// TwinCAT 3 PLC project PLC1
// ProgramVersion: 3.1.4024.0
// libraries:
//   Tc2_Standard, * (Beckhoff Automation GmbH)
//   Tc2_System, * (Beckhoff Automation GmbH)
//   Tc3_Module, * (Beckhoff Automation GmbH)
// project tree:
//   / PlcTask.TcTTO
//   POUs/ ContactorNO.TcPOU, LedLamp.TcPOU, MAIN.TcPOU, StartButton.TcPOU
// real-time tasks:
//   TASK PlcTask: cycle T#10ms, priority 20, ADS port 350

CONFIGURATION PLC1
    RESOURCE PLC ON TwinCAT3
        TASK PlcTask(INTERVAL := T#10ms, PRIORITY := 20);
        PROGRAM MAIN WITH PlcTask : MAIN;
    END_RESOURCE
END_CONFIGURATION

// ---- POUs/MAIN.TcPOU
PROGRAM MAIN
VAR
	startButton : StartButton;
END_VAR

startButton();

END_PROGRAM

// ---- POUs/StartButton.TcPOU
FUNCTION_BLOCK StartButton
VAR
	input AT %I* : BOOL;
END_VAR

PROPERTY IsPressed : BOOL
GET
IsPressed := input
END_GET
END_PROPERTY

PROPERTY IsReleased : BOOL
GET
IsReleased := NOT input;
END_GET
END_PROPERTY

END_FUNCTION_BLOCK

// ---- POUs/ContactorNO.TcPOU
FUNCTION_BLOCK ContactorNO
VAR
	output AT %Q* : BOOL;
END_VAR

METHOD Close
VAR_INPUT
END_VAR
output := TRUE;
END_METHOD

PROPERTY IsClose : BOOL
GET
IsClose := output;
END_GET
END_PROPERTY

PROPERTY IsOpen : BOOL
GET
IsOpen := NOT output;
END_GET
END_PROPERTY

METHOD Open
VAR_INPUT
END_VAR
output := FALSE;
END_METHOD

END_FUNCTION_BLOCK

// ---- POUs/LedLamp.TcPOU
FUNCTION_BLOCK LedLamp
VAR
	output AT %Q* : BOOL;
END_VAR

METHOD Off
VAR_INPUT
END_VAR
output := FALSE;
END_METHOD

METHOD On
VAR_INPUT
END_VAR
output := TRUE;
END_METHOD

END_FUNCTION_BLOCK
